(* LS Electric XG5000 project: LoadCell_LD02S_Sample *)
(* PLC LSPLC *)
(* module base 0 slot 0: Input/Output Module:XEM-DN/DP32HP (DC 24V Input, Transistor Output, 32 Contacts) *)
(* module base 0 slot 1: Internal Positioning:XBF-PO06E (Open Collector Type, 6 Axis) *)
(* module base 0 slot 2: Loadcell Input Module:XBF-LD02S (Isolated-type Loadcell Input(2 Channels)) *)
VAR_GLOBAL
    _02_CH0_ERR AT %UX0.2.30 : BOOL; (* Loadcell Input Module: CH0 Error *)
    _02_CH0_GWDATA AT %UD0.2.3 : DINT; (* Loadcell Input Module: CH0  Gross Weight Data *)
    _02_CH0_GWMAX AT %UD0.2.9 : DWORD; (* Loadcell Input Module: CH0 Gross Weight Max. Data *)
    _02_CH0_GWMIN AT %UD0.2.10 : DWORD; (* Loadcell Input Module: CH0 Gross Weight Min. Data *)
    _02_CH0_RUN AT %UX0.2.16 : BOOL; (* Loadcell Input Module: CH0 Run Status *)
    _02_CH1_ERR AT %UX0.2.31 : BOOL; (* Loadcell Input Module: CH1 Error *)
    _02_CH1_GWDATA AT %UD0.2.4 : DINT; (* Loadcell Input Module: CH1 Gross Weight Data *)
    _02_CH1_GWMAX AT %UD0.2.11 : DWORD; (* Loadcell Input Module: CH1 Gross Weight Max. Data *)
    _02_CH1_GWMIN AT %UD0.2.12 : DWORD; (* Loadcell Input Module: CH1 Gross Weight Min. Data *)
    _02_CH1_RUN AT %UX0.2.17 : BOOL; (* Loadcell Input Module: CH1 Run Status *)
    _02_RDY AT %UX0.2.15 : BOOL; (* Loadcell Input Module: Ready Flag *)
END_VAR

(* Comments on direct variables
%MX0	Comment 0
%MX1	Comment 1
%MX2	Comment 2
%MX3	Comment 3
%MX4	Comment 4
%MX5	Comment 5
%MX6	Comment 6
%MX7	Comment 7
%MX8	Comment 0
%MX9	Comment 0
%MX10	Comment 0
%MX11	Comment 0
%MX12	Comment 0
%MX13	Comment 0
%MX14	Comment 0
%MX15	Comment 0
%MX16	Comment 0
%MX17	Comment 0
%MX18	Comment 0
%MX19	Comment 0
%MX20	Comment 0
%MX21	Comment 0
%MX22	Comment 0
%MX23	Comment 0
%MX24	Comment 0
%MX25	Comment 0
%MX26	Comment 0
%MX27	Comment 0
%MX28	Comment 0
%MX29	Comment 0
*)

PROGRAM SampleLoadCell (* task: Scan Program *)
(* sample code for load cell LD02S *)
VAR
    CH0_Gross_Weight : DINT; (* Gross weight value of CH0 *)
    CH1_Gross_Weight : DINT; (* Gross weight value of CH1 *)
    Store_CH0_GrossWeightData : BOOL; (* Flag to store gross weight data from CH0 *)
    Store_CH1_GrossWeightData : BOOL; (* flag to store gross weight data from CH1 *)
END_VAR
VAR_EXTERNAL
    _02_CH0_ERR : BOOL; (* AT %UX0.2.30 *) (* Loadcell Input Module: CH0 Error *)
    _02_CH0_GWDATA : DINT; (* AT %UD0.2.3 *) (* Loadcell Input Module: CH0  Gross Weight Data *)
    _02_CH0_GWMAX : DWORD; (* AT %UD0.2.9 *) (* Loadcell Input Module: CH0 Gross Weight Max. Data *)
    _02_CH0_GWMIN : DWORD; (* AT %UD0.2.10 *) (* Loadcell Input Module: CH0 Gross Weight Min. Data *)
    _02_CH0_RUN : BOOL; (* AT %UX0.2.16 *) (* Loadcell Input Module: CH0 Run Status *)
    _02_CH1_ERR : BOOL; (* AT %UX0.2.31 *) (* Loadcell Input Module: CH1 Error *)
    _02_CH1_GWDATA : DINT; (* AT %UD0.2.4 *) (* Loadcell Input Module: CH1 Gross Weight Data *)
    _02_CH1_GWMAX : DWORD; (* AT %UD0.2.11 *) (* Loadcell Input Module: CH1 Gross Weight Max. Data *)
    _02_CH1_GWMIN : DWORD; (* AT %UD0.2.12 *) (* Loadcell Input Module: CH1 Gross Weight Min. Data *)
    _02_CH1_RUN : BOOL; (* AT %UX0.2.17 *) (* Loadcell Input Module: CH1 Run Status *)
    _02_RDY : BOOL; (* AT %UX0.2.15 *) (* Loadcell Input Module: Ready Flag *)
END_VAR

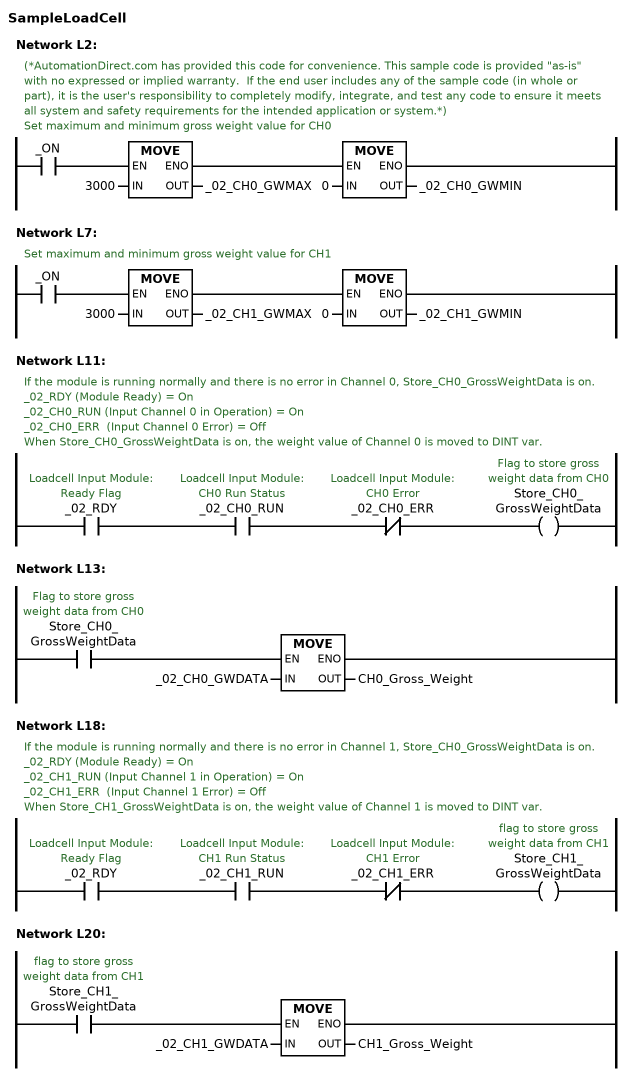
(* ( *AutomationDirect.com has provided this code for convenience. This sample code is provided "as-is" with no expressed or implied warranty.  If the end user includes any of the sample code (in whole or part), it is the user's responsibility to completely modify, integrate, and test any code to ensure it meets all system and safety requirements for the intended application or system.* ) *)
(* Set maximum and minimum gross weight value for CH0 *)
(* Rung L2 *)
IF _ON THEN
    _02_CH0_GWMAX := 3000;
    _02_CH0_GWMIN := 0;
END_IF;
(* Set maximum and minimum gross weight value for CH1 *)
(* Rung L7 *)
IF _ON THEN
    _02_CH1_GWMAX := 3000;
    _02_CH1_GWMIN := 0;
END_IF;
(* If the module is running normally and there is no error in Channel 0, Store_CH0_GrossWeightData is on. / _02_RDY (Module Ready) = On / _02_CH0_RUN (Input Channel 0 in Operation) = On / _02_CH0_ERR  (Input Channel 0 Error) = Off / When Store_CH0_GrossWeightData is on, the weight value of Channel 0 is moved to DINT var. *)
(* Rung L11 *)
Store_CH0_GrossWeightData := _02_RDY AND _02_CH0_RUN AND NOT _02_CH0_ERR;
(* Rung L13 *)
IF Store_CH0_GrossWeightData THEN CH0_Gross_Weight := _02_CH0_GWDATA; END_IF;
(* If the module is running normally and there is no error in Channel 1, Store_CH0_GrossWeightData is on. / _02_RDY (Module Ready) = On / _02_CH1_RUN (Input Channel 1 in Operation) = On / _02_CH1_ERR  (Input Channel 1 Error) = Off / When Store_CH1_GrossWeightData is on, the weight value of Channel 1 is moved to DINT var. *)
(* Rung L18 *)
Store_CH1_GrossWeightData := _02_RDY AND _02_CH1_RUN AND NOT _02_CH1_ERR;
(* Rung L20 *)
IF Store_CH1_GrossWeightData THEN CH1_Gross_Weight := _02_CH1_GWDATA; END_IF;
END_PROGRAM